PROGRAM HMI
VAR
END_VAR

IF GVL.appRUN = FALSE AND GVL.noFaultDetected = TRUE THEN 
	GVL.chargeCOIL := HMI_DB.ActivateChargePB;
	GVL.softdump 	:= HMI_DB.ActivateDumpPB;
	END_IF
	
//FAULTS - Underdevelopment

HMI_DB.Fault.0 := GVL.sparkdetect;
HMI_DB.Fault.1 := GVL.FireDetected;

//HMI_DB.Fault.2 := 
//HMI_DB.Fault.3 := 

//TRIPS



//PERMISSIVES


//HMI bit mapping
HMI_DB.Charging := GVL.chargeCOIL_contact;
HMI_DB.Dumping := NOT GVL.softdump_contact;

(*IF GVL.softdump_contact = FALSE THEN  //softdump_contact is normally closed.  When closed, dumping coil is open.
	HMI_DB.Dumping := TRUE;
ELSE
	HMI_DB.Dumping := FALSE;
END_IF;*)

END_PROGRAM

(* stored: Version 1.1.0.1, ProductVersion 3.1.4024.9
   POU HMI: Id {dc100eb0-1044-40f8-af7c-fa22d9cf173d}, SpecialFunc None *)
